// TIA Portal V20 export
TYPE "MaxMin"
   STRUCT
      Min : Real;
      Max : Real;
   END_STRUCT;
END_TYPE
